{attribute addProperty BoxType "EL3102--0000"}
{attribute addProperty Id "StatusAT %I*BYTE811ValueAT %I*INT1622"}
{attribute addProperty CRC "2721721305"}
{attribute addProperty SizeInBites "24"}
{attribute addProperty SizeInBytes "3"}
TYPE Channel_A23A2BD9 :
STRUCT
	{attribute addProperty Name "Status"}
	Status AT %I* : BYTE;
	{attribute addProperty Name "Value"}
	Value AT %I* : INT;
END_STRUCT
END_TYPE

(* stored: Version 1.2.0.0, ProductVersion 3.1.4024.9
   DUT Channel_A23A2BD9: Id {1811cdd9-36b6-4f99-a276-f865ff4deb85} *)
